{attribute 'qualified_only'}
{attribute 'strict'}
TYPE EventLevel :
(
	INFO := 10,
  WARNING :=20,
  ERROR := 30
) BYTE := INFO;
END_TYPE

(* stored: Version 1.1.0.1, ProductVersion 3.1.4024.9
   DUT EventLevel: Id {ca81352f-d08f-465b-acbe-efc11506cc1d} *)
